# EPICS autosave request: iocBoot/sioc-sps-im01/sioc-sps-im01.req
file "lcls2.req" AREA=SPS,POS=605
